KUKA KRL program: rtestegarra.src, rtestegarra.dat

--- rtestegarra.src ---
&ACCESS RVP
&REL 2
&COMMENT Teste da Garra
DEF rTesteGarra ( )
;Routine to check the gripper
;
;Stop $Advance
nMemoAdvance=$ADVANCE
$ADVANCE=0

;Clear generic counter
I[20]=0

;Start routine
$OUT[358]=TRUE

;Close and open gripper to perform check
;
rFechaGarra()
;
rAbreGarra(GARRA_1_E_2)
;
rFechaGarra()

;Returns $Advance
$ADVANCE=nMemoAdvance

;End of routine
$OUT[358]=FALSE

END

--- rtestegarra.dat ---
&ACCESS RVP
&REL 2
&COMMENT Teste da Garra
DEFDAT rTesteGarra PUBLIC
;FOLD EXTERNAL DECLARATIONS;%{PE}%MKUKATPBASIS,%CEXT,%VCOMMON,%P
;FOLD BASISTECH EXT;%{PE}%MKUKATPBASIS,%CEXT,%VEXT,%P
EXT  BAS (BAS_COMMAND  :IN,REAL  :IN )
DECL INT SUCCESS
;ENDFOLD (BASISTECH EXT)
;FOLD USER EXT;%{E}%MKUKATPUSER,%CEXT,%VEXT,%P
;Make here your modifications

;ENDFOLD (USER EXT)
;ENDFOLD (EXTERNAL DECLERATIONS)
ENDDAT
